FUNCTION_BLOCK MixerLogic (* CAT Function Block Type *)
  (* Standard: 61499-2 *)
  (* Version 0.0, 6/15/2026, Schneider Electric, template *)
  PACKAGE SE.Nereda;
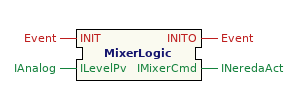
  EVENT_INPUT
    INIT;
  END_EVENT
  EVENT_OUTPUT
    INITO;
  END_EVENT
  SOCKETS
    ILevelPv : IAnalog;
  END_SOCKETS
  PLUGS
    IMixerCmd : INeredaAct;
  END_PLUGS
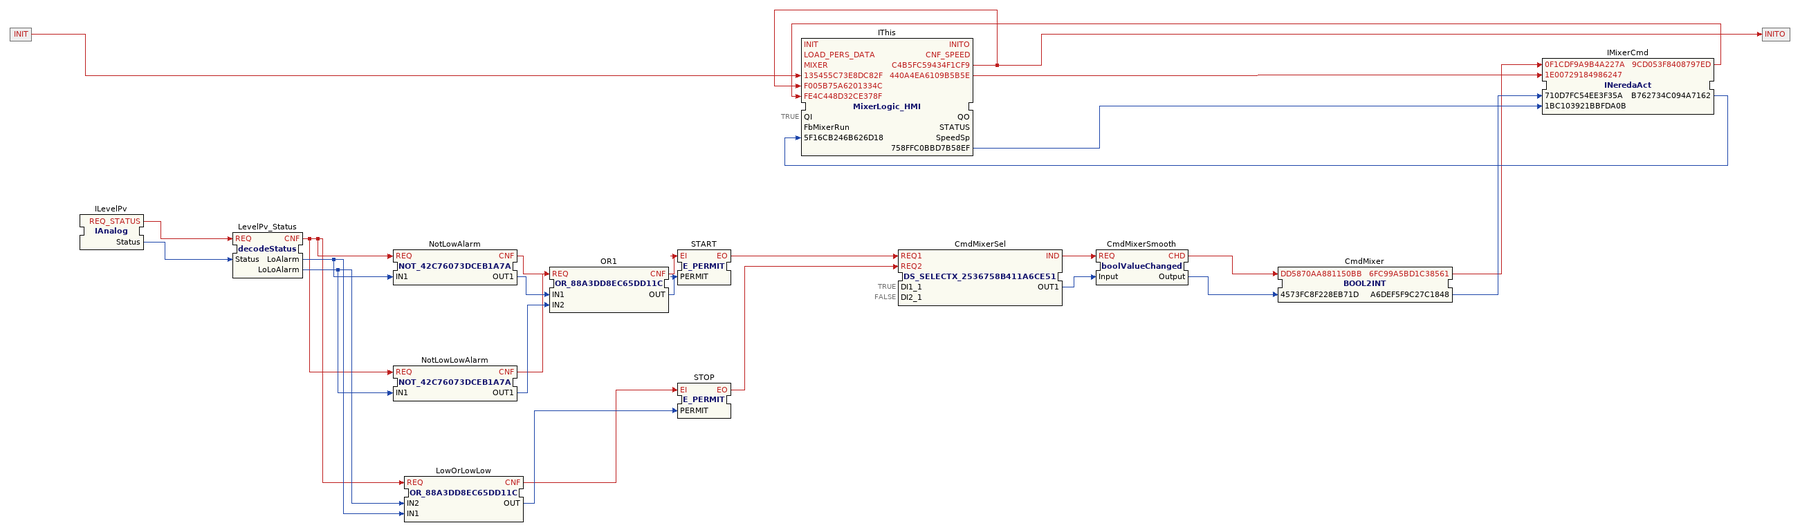
  (* 01 - FUNCTIONNAL INPUT INTERFACE *)
  (* 00 - INITIALIZATION *)
  (* 05 - LOGIC *)
  (* 06 - HMI INTERFACE *)
  (* 03 - FIELD INTERFACE *)
  (* Mixer Logic *)
  (* 02 - FUNCTIONNAL OUTPUT INTERFACE *)
  FBS
    LevelPv_Status : decodeStatus;
    IThis : MixerLogic_HMI(QI := TRUE);
    START : E_PERMIT;
    STOP : E_PERMIT;
    NotLowAlarm : NOT_42C76073DCEB1A7A; {SET_ATTRIBUTE(Configuration.GenericFBType.InterfaceParams, Runtime.Standard#CNT:=1;OUT${CNT$}:BOOL)}
    CmdMixerSel : DS_SELECTX_2536758B411A6CE51(DI1_1 := TRUE, DI2_1 := FALSE); {SET_ATTRIBUTE(Configuration.GenericFBType.InterfaceParams, Runtime.Standard#CNTX:=2;CNTY:=1;DI${CNTX,_,CNTY$}:BOOL)}
    CmdMixerSmooth : boolValueChanged;
    CmdMixer : BOOL2INT;
    OR1 : OR_88A3DD8EC65DD11C; {SET_ATTRIBUTE(Configuration.GenericFBType.InterfaceParams, Runtime.Standard#CNT:=2;OUT:BOOL)}
    NotLowLowAlarm : NOT_42C76073DCEB1A7A; {SET_ATTRIBUTE(Configuration.GenericFBType.InterfaceParams, Runtime.Standard#CNT:=1;OUT${CNT$}:BOOL)}
    LowOrLowLow : OR_88A3DD8EC65DD11C; {SET_ATTRIBUTE(Configuration.GenericFBType.InterfaceParams, Runtime.Standard#CNT:=2;OUT:BOOL)}
  END_FBS
  EVENT_CONNECTIONS
    ILevelPv.REQ_STATUS TO LevelPv_Status.REQ;
    LevelPv_Status.CNF TO NotLowAlarm.REQ;
    LevelPv_Status.CNF TO LowOrLowLow.REQ;
    NotLowAlarm.CNF TO OR1.REQ;
    START.EO TO CmdMixerSel.REQ1;
    CmdMixerSel.IND TO CmdMixerSmooth.REQ;
    STOP.EO TO CmdMixerSel.REQ2;
    CmdMixerSmooth.CHD TO CmdMixer.DD5870AA881150BB;
    CmdMixer.6FC99A5BD1C38561 TO IMixerCmd.0F1CDF9A9B4A227A;
    INIT TO IThis.135455C73E8DC82F;
    IThis.C4B5FC59434F1CF9 TO IThis.F005B75A6201334C;
    IMixerCmd.9CD053F8408797ED TO IThis.FE4C448D32CE378F;
    IThis.C4B5FC59434F1CF9 TO INITO;
    IThis.440A4EA6109B5B5E TO IMixerCmd.1E00729184986247;
    OR1.CNF TO START.EI;
    LevelPv_Status.CNF TO NotLowLowAlarm.REQ;
    NotLowLowAlarm.CNF TO OR1.REQ;
    LowOrLowLow.CNF TO STOP.EI;
  END_CONNECTIONS
  DATA_CONNECTIONS
    ILevelPv.Status TO LevelPv_Status.Status;
    NotLowAlarm.OUT1 TO OR1.IN1;
    LevelPv_Status.LoAlarm TO NotLowAlarm.IN1;
    CmdMixerSel.OUT1 TO CmdMixerSmooth.Input;
    CmdMixerSmooth.Output TO CmdMixer.4573FC8F228EB71D;
    CmdMixer.A6DEF5F9C27C1848 TO IMixerCmd.710D7FC54EE3F35A;
    IThis.758FFC0BBD7B58EF TO IMixerCmd.1BC103921BBFDA0B;
    IMixerCmd.B762734C094A7162 TO IThis.5F16CB246B626D18;
    LevelPv_Status.LoLoAlarm TO LowOrLowLow.IN2;
    NotLowLowAlarm.OUT1 TO OR1.IN2;
    OR1.OUT TO START.PERMIT;
    LowOrLowLow.OUT TO STOP.PERMIT;
    LevelPv_Status.LoLoAlarm TO NotLowLowAlarm.IN1;
    LevelPv_Status.LoAlarm TO LowOrLowLow.IN1;
  END_CONNECTIONS
END_FUNCTION_BLOCK
